PROGRAM test
VAR
	xTestInput	AT %I* : BOOL;
END_VAR

END_PROGRAM

(* stored: Version 1.1.0.1, ProductVersion 3.1.4024.9
   POU test: Id {041284d1-4032-4a04-9824-3e720f32b5ff}, SpecialFunc None *)
